// TIA Portal project "六路温湿度采集" (V16)

(* hardware
DEVICE "S71500/ET200MP station_1"  S7-1500 station
   slot 0: "导轨_0"  Rack  6ES7 590-1***0-0AA0
   slot 1: "PLC_1"  CPU 1512C-1 PN  6ES7 512-1CK01-0AB0  V2.8
      slot 3: "CPU 显示_1"  6ES7591-1AA00-0AA0
      slot 32768: "PROFINET 接口_1"  X1
         slot 32769: "端口_1"  X1 P1
         slot 32770: "端口_2"  X1 P2
      slot 34817: "Virtual CP interface port_1"  Virtual CP interface port  Virtual CP interface port
*)

// ===== PLC "PLC_1"  CPU 1512C-1 PN =====

VAR_GLOBAL   // PLC tag table "默认变量表"
   "中间变量" AT %MW100 : Word;
   "Tag_1" AT %M0.0 : Bool;
   "System_Byte" AT %MB1 : Byte;
   "FirstScan" AT %M1.0 : Bool;
   "DiagStatusUpdate" AT %M1.1 : Bool;
   "AlwaysTRUE" AT %M1.2 : Bool;
   "AlwaysFALSE" AT %M1.3 : Bool;
   "Tag_2" AT %M2.0 : Bool;
END_VAR

DATA_BLOCK "ModbusTCPData"   // DB1
{ S7_Optimized_Access := 'FALSE' }
VERSION : 0.1
   VAR
      模块1温度 : Int;
      模块1湿度 : Int;
      模块2温度 : Int;
      模块2湿度 : Int;
      模块3温度 : Int;
      模块3湿度 : Int;
      模块4温度 : Int;
      模块4湿度 : Int;
      模块5温度 : Int;
      模块5湿度 : Int;
      模块6温度 : Int;
      模块6湿度 : Int;
      模块1温度高 : Bool;
      模块1温度低 : Bool;
      模块1湿度高 : Bool;
      模块1湿度低 : Bool;
      模块1异常 : Bool;
      空1 : Bool;
      空2 : Bool;
      空3 : Bool;
      空byte1 : Byte;
      模块2温度高 : Bool;
      模块2温度低 : Bool;
      模块2湿度高 : Bool;
      模块2湿度低 : Bool;
      模块2异常 : Bool;
      空4 : Bool;
      空5 : Bool;
      空6 : Bool;
      空byte2 : Byte;
      模块3温度高 : Bool;
      模块3温度低 : Bool;
      模块3湿度高 : Bool;
      模块3湿度低 : Bool;
      模块3异常 : Bool;
      空7 : Bool;
      空8 : Bool;
      空9 : Bool;
      空byte3 : Byte;
      模块4温度高 : Bool;
      模块4温度低 : Bool;
      模块4湿度高 : Bool;
      模块4湿度低 : Bool;
      模块4异常 : Bool;
      空11 : Bool;
      空12 : Bool;
      空13 : Bool;
      空byte4 : Byte;
      模块5温度高 : Bool;
      模块5温度低 : Bool;
      模块5湿度高 : Bool;
      模块5湿度低 : Bool;
      模块5异常 : Bool;
      空14 : Bool;
      空15 : Bool;
      空16 : Bool;
      空byte5 : Byte;
      模块6温度高 : Bool;
      模块6温度低 : Bool;
      模块6湿度高 : Bool;
      模块6湿度低 : Bool;
      模块6异常 : Bool;
      空byte6 : Byte;
      模块1温度高限 : Int := 35;
      模块1温度低限 : Int := 25;
      模块1湿度高限 : Int := 25;
      模块1湿度低限 : Int := 15;
      模块2温度高限 : Int := 35;
      模块2温度低限 : Int := 25;
      模块2湿度高限 : Int := 25;
      模块2湿度低限 : Int := 15;
      模块3温度高限 : Int := 35;
      模块3温度低限 : Int := 25;
      模块3湿度高限 : Int := 25;
      模块3湿度低限 : Int := 15;
      模块4温度高限 : Int := 35;
      模块4温度低限 : Int := 25;
      模块4湿度高限 : Int := 25;
      模块4湿度低限 : Int := 15;
      模块5温度高限 : Int := 35;
      模块5温度低限 : Int := 25;
      模块5湿度高限 : Int := 25;
      模块5湿度低限 : Int := 15;
      模块6温度高限 : Int := 35;
      模块6温度低限 : Int := 25;
      模块6湿度高限 : Int := 25;
      模块6湿度低限 : Int := 15;
      模块1温度报警启用 : Int := 0;
      模块1湿度报警启用 : Int;
      模块2温度报警启用 : Int;
      模块2湿度报警启用 : Int;
      模块3温度报警启用 : Int;
      模块3湿度报警启用 : Int;
      模块4温度报警启用 : Int;
      模块4湿度报警启用 : Int;
      模块5温度报警启用 : Int;
      模块5湿度报警启用 : Int;
      模块6温度报警启用 : Int;
      模块6湿度报警启用 : Int;
      串口站地址 : Int;
      串口波特率 : Int;
      "IP地址-1" : Int;
      "IP地址-2" : Int;
      "IP地址-3" : Int;
      "IP地址-4" : Int;
      以太网端口号 : Int;
      "以太网参数写入确认（PC写1）" : Int;
   END_VAR
BEGIN
END_DATA_BLOCK

DATA_BLOCK "通信参数的DB块"   // DB3
{ S7_Optimized_Access := 'TRUE' }
VERSION : 0.1
   VAR
      Conn : TCON_IP_v4;
   END_VAR
BEGIN
   Conn.InterfaceId := 64;
   Conn.ID := 1;
   Conn.LocalPort := 502;
END_DATA_BLOCK

DATA_BLOCK "DateTime"   // DB4
{ S7_Optimized_Access := 'TRUE' }
VERSION : 0.1
   VAR
      day_time : DTL;
      ReadDateTIme_Now : Int;
   END_VAR
BEGIN
END_DATA_BLOCK

FUNCTION "温湿度模块超限报警" : Void   // FC1, LAD
{ S7_Optimized_Access := 'TRUE' }
VERSION : 0.1
   VAR_INPUT
      模块温度 : Int;
      模块温度高限 : Int;
      模块温度低限 : Int;
      模块湿度 : Int;
      模块湿度高限 : Int;
      模块湿度低限 : Int;
      模块温度报警启用 : Int;
      模块湿度报警启用 : Int;
   END_VAR
   VAR_OUTPUT
      模块异常 : Bool;
   END_VAR
   VAR_IN_OUT
      模块温度高 : Bool;
      模块温度低 : Bool;
      模块湿度高 : Bool;
      模块湿度低 : Bool;
   END_VAR
   VAR_TEMP   // added for the SCL form of the ladder/FBD networks
      _w1 : Bool;
      _w2 : Bool;
   END_VAR
BEGIN

REGION Network 1
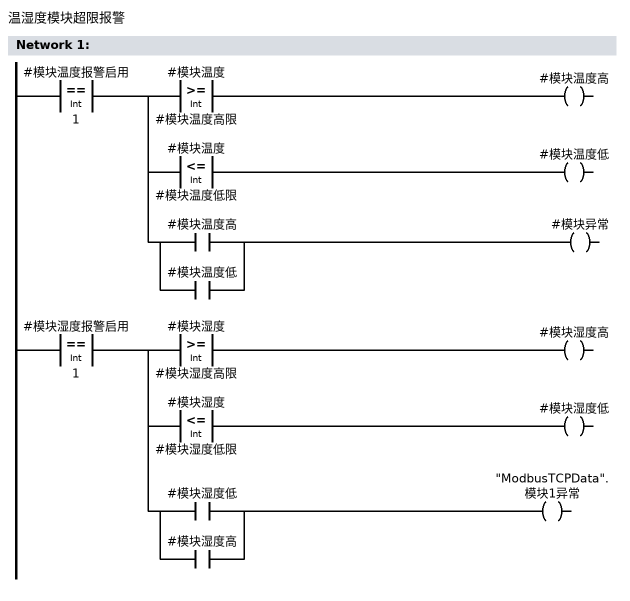
   RUNG wire#powerrail
      { S7_Templates := "SrcType := Int" } EQ_Contact(in1 := #模块温度报警启用, in2 := 1)
      wire#w1
      { S7_Templates := "SrcType := Int" } GE_Contact(in1 := #模块温度, in2 := #模块温度高限)
      Coil( #模块温度高 )
   END_RUNG
   RUNG wire#w1
      { S7_Templates := "SrcType := Int" } LE_Contact(in1 := #模块温度, in2 := #模块温度低限)
      Coil( #模块温度低 )
   END_RUNG
   RUNG wire#w1
      Contact( #模块温度高 )
      wire#w2
      Coil( #模块异常 )
   END_RUNG
   RUNG wire#w1
      Contact( #模块温度低 )
   END_RUNG wire#w2
   RUNG wire#powerrail
      { S7_Templates := "SrcType := Int" } EQ_Contact(in1 := #模块湿度报警启用, in2 := 1)
      wire#w3
      { S7_Templates := "SrcType := Int" } GE_Contact(in1 := #模块湿度, in2 := #模块湿度高限)
      Coil( #模块湿度高 )
   END_RUNG
   RUNG wire#w3
      { S7_Templates := "SrcType := Int" } LE_Contact(in1 := #模块湿度, in2 := #模块湿度低限)
      Coil( #模块湿度低 )
   END_RUNG
   RUNG wire#w3
      Contact( #模块湿度低 )
      wire#w4
      Coil( "ModbusTCPData".模块1异常 )
   END_RUNG
   RUNG wire#w3
      Contact( #模块湿度高 )
   END_RUNG wire#w4
   // the same network as SCL:
   #_w1 := #模块温度报警启用 = 1;
   #模块温度高 := #_w1 AND (#模块温度 >= #模块温度高限);
   #模块温度低 := #_w1 AND (#模块温度 <= #模块温度低限);
   #模块异常 := #_w1 AND (#模块温度高 OR #模块温度低);
   #_w2 := #模块湿度报警启用 = 1;
   #模块湿度高 := #_w2 AND (#模块湿度 >= #模块湿度高限);
   #模块湿度低 := #_w2 AND (#模块湿度 <= #模块湿度低限);
   "ModbusTCPData".模块1异常 := #_w2 AND (#模块湿度低 OR #模块湿度高);
END_REGION
END_FUNCTION

ORGANIZATION_BLOCK "Main"   // OB1, LAD, ProgramCycle
TITLE = "Main Program Sweep (Cycle)"
{ S7_Optimized_Access := 'TRUE' }
VERSION : 0.1
   VAR_INPUT
      Initial_Call : Bool;   // Initial call of this OB
      Remanence : Bool;   // =True, if remanent data are available
   END_VAR
BEGIN

REGION Network 1: 设定PLC的客户端，通信的变量
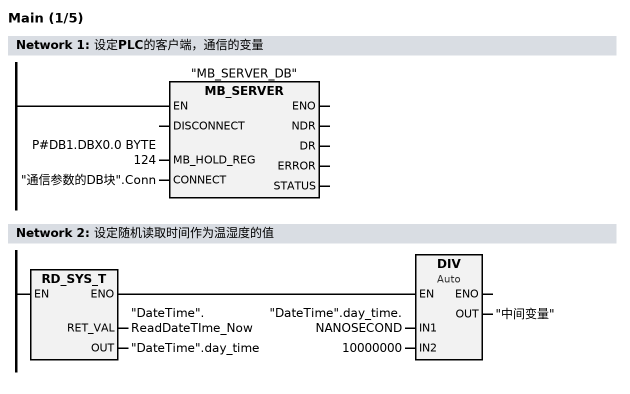
   "MB_SERVER_DB"(MB_HOLD_REG := P#DB1.DBX0.0 BYTE 124, CONNECT := "通信参数的DB块".Conn);   // MB_SERVER
END_REGION

REGION Network 2: 设定随机读取时间作为温湿度的值
   // ENO of a box is taken as its EN; it also drops when the box reports an error
   "DateTime".ReadDateTIme_Now := RD_SYS_T(OUT => "DateTime".day_time);
   "中间变量" := "DateTime".day_time.NANOSECOND / 10000000;
END_REGION

REGION Network 3: 将随机时间传递六路温湿度
   // 因为是毫秒机的显示，所以可以保证每个都不相同
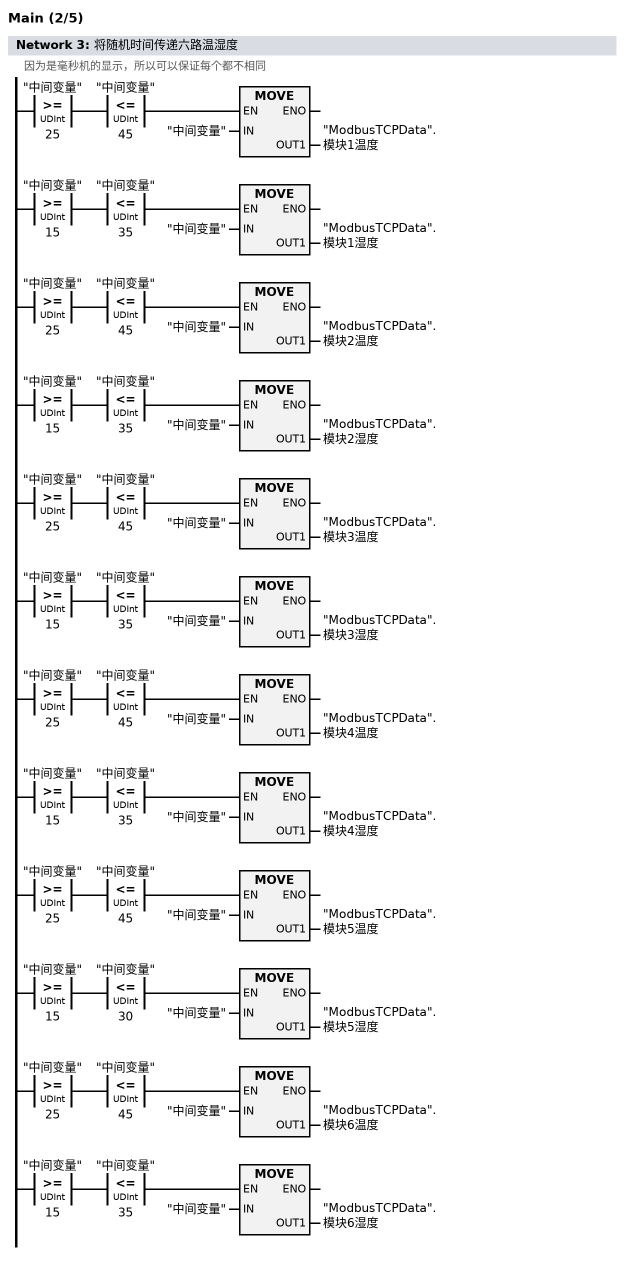
   RUNG wire#powerrail
      { S7_Templates := "SrcType := UDInt" } GE_Contact(in1 := "中间变量", in2 := 25)
      { S7_Templates := "SrcType := UDInt" } LE_Contact(in1 := "中间变量", in2 := 45)
      Move(in := "中间变量", out1 => "ModbusTCPData".模块1温度)
   END_RUNG
   RUNG wire#powerrail
      { S7_Templates := "SrcType := UDInt" } GE_Contact(in1 := "中间变量", in2 := 15)
      { S7_Templates := "SrcType := UDInt" } LE_Contact(in1 := "中间变量", in2 := 35)
      Move(in := "中间变量", out1 => "ModbusTCPData".模块1湿度)
   END_RUNG
   RUNG wire#powerrail
      { S7_Templates := "SrcType := UDInt" } GE_Contact(in1 := "中间变量", in2 := 25)
      { S7_Templates := "SrcType := UDInt" } LE_Contact(in1 := "中间变量", in2 := 45)
      Move(in := "中间变量", out1 => "ModbusTCPData".模块2温度)
   END_RUNG
   RUNG wire#powerrail
      { S7_Templates := "SrcType := UDInt" } GE_Contact(in1 := "中间变量", in2 := 15)
      { S7_Templates := "SrcType := UDInt" } LE_Contact(in1 := "中间变量", in2 := 35)
      Move(in := "中间变量", out1 => "ModbusTCPData".模块2湿度)
   END_RUNG
   RUNG wire#powerrail
      { S7_Templates := "SrcType := UDInt" } GE_Contact(in1 := "中间变量", in2 := 25)
      { S7_Templates := "SrcType := UDInt" } LE_Contact(in1 := "中间变量", in2 := 45)
      Move(in := "中间变量", out1 => "ModbusTCPData".模块3温度)
   END_RUNG
   RUNG wire#powerrail
      { S7_Templates := "SrcType := UDInt" } GE_Contact(in1 := "中间变量", in2 := 15)
      { S7_Templates := "SrcType := UDInt" } LE_Contact(in1 := "中间变量", in2 := 35)
      Move(in := "中间变量", out1 => "ModbusTCPData".模块3湿度)
   END_RUNG
   RUNG wire#powerrail
      { S7_Templates := "SrcType := UDInt" } GE_Contact(in1 := "中间变量", in2 := 25)
      { S7_Templates := "SrcType := UDInt" } LE_Contact(in1 := "中间变量", in2 := 45)
      Move(in := "中间变量", out1 => "ModbusTCPData".模块4温度)
   END_RUNG
   RUNG wire#powerrail
      { S7_Templates := "SrcType := UDInt" } GE_Contact(in1 := "中间变量", in2 := 15)
      { S7_Templates := "SrcType := UDInt" } LE_Contact(in1 := "中间变量", in2 := 35)
      Move(in := "中间变量", out1 => "ModbusTCPData".模块4湿度)
   END_RUNG
   RUNG wire#powerrail
      { S7_Templates := "SrcType := UDInt" } GE_Contact(in1 := "中间变量", in2 := 25)
      { S7_Templates := "SrcType := UDInt" } LE_Contact(in1 := "中间变量", in2 := 45)
      Move(in := "中间变量", out1 => "ModbusTCPData".模块5温度)
   END_RUNG
   RUNG wire#powerrail
      { S7_Templates := "SrcType := UDInt" } GE_Contact(in1 := "中间变量", in2 := 15)
      { S7_Templates := "SrcType := UDInt" } LE_Contact(in1 := "中间变量", in2 := 30)
      Move(in := "中间变量", out1 => "ModbusTCPData".模块5湿度)
   END_RUNG
   RUNG wire#powerrail
      { S7_Templates := "SrcType := UDInt" } GE_Contact(in1 := "中间变量", in2 := 25)
      { S7_Templates := "SrcType := UDInt" } LE_Contact(in1 := "中间变量", in2 := 45)
      Move(in := "中间变量", out1 => "ModbusTCPData".模块6温度)
   END_RUNG
   RUNG wire#powerrail
      { S7_Templates := "SrcType := UDInt" } GE_Contact(in1 := "中间变量", in2 := 15)
      { S7_Templates := "SrcType := UDInt" } LE_Contact(in1 := "中间变量", in2 := 35)
      Move(in := "中间变量", out1 => "ModbusTCPData".模块6湿度)
   END_RUNG
   // the same network as SCL:
   IF ("中间变量" >= 25) AND ("中间变量" <= 45) THEN "ModbusTCPData".模块1温度 := "中间变量"; END_IF;
   IF ("中间变量" >= 15) AND ("中间变量" <= 35) THEN "ModbusTCPData".模块1湿度 := "中间变量"; END_IF;
   IF ("中间变量" >= 25) AND ("中间变量" <= 45) THEN "ModbusTCPData".模块2温度 := "中间变量"; END_IF;
   IF ("中间变量" >= 15) AND ("中间变量" <= 35) THEN "ModbusTCPData".模块2湿度 := "中间变量"; END_IF;
   IF ("中间变量" >= 25) AND ("中间变量" <= 45) THEN "ModbusTCPData".模块3温度 := "中间变量"; END_IF;
   IF ("中间变量" >= 15) AND ("中间变量" <= 35) THEN "ModbusTCPData".模块3湿度 := "中间变量"; END_IF;
   IF ("中间变量" >= 25) AND ("中间变量" <= 45) THEN "ModbusTCPData".模块4温度 := "中间变量"; END_IF;
   IF ("中间变量" >= 15) AND ("中间变量" <= 35) THEN "ModbusTCPData".模块4湿度 := "中间变量"; END_IF;
   IF ("中间变量" >= 25) AND ("中间变量" <= 45) THEN "ModbusTCPData".模块5温度 := "中间变量"; END_IF;
   IF ("中间变量" >= 15) AND ("中间变量" <= 30) THEN "ModbusTCPData".模块5湿度 := "中间变量"; END_IF;
   IF ("中间变量" >= 25) AND ("中间变量" <= 45) THEN "ModbusTCPData".模块6温度 := "中间变量"; END_IF;
   IF ("中间变量" >= 15) AND ("中间变量" <= 35) THEN "ModbusTCPData".模块6湿度 := "中间变量"; END_IF;
END_REGION

REGION Network 4
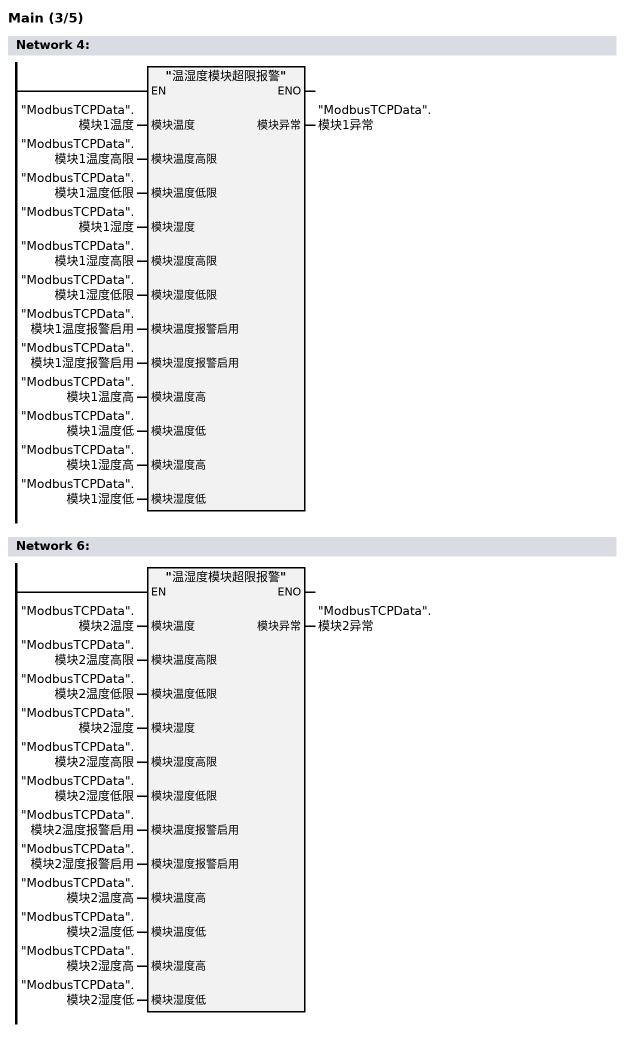
   RUNG wire#powerrail
      "温湿度模块超限报警"(模块温度 := "ModbusTCPData".模块1温度, 模块温度高限 := "ModbusTCPData".模块1温度高限, 模块温度低限 := "ModbusTCPData".模块1温度低限, 模块湿度 := "ModbusTCPData".模块1湿度, 模块湿度高限 := "ModbusTCPData".模块1湿度高限, 模块湿度低限 := "ModbusTCPData".模块1湿度低限, 模块温度报警启用 := "ModbusTCPData".模块1温度报警启用, 模块湿度报警启用 := "ModbusTCPData".模块1湿度报警启用, 模块温度高 := "ModbusTCPData".模块1温度高, 模块温度低 := "ModbusTCPData".模块1温度低, 模块湿度高 := "ModbusTCPData".模块1湿度高, 模块湿度低 := "ModbusTCPData".模块1湿度低, 模块异常 => "ModbusTCPData".模块1异常)
   END_RUNG
   // the same network as SCL:
   "温湿度模块超限报警"(模块温度 := "ModbusTCPData".模块1温度,
               模块温度高限 := "ModbusTCPData".模块1温度高限,
               模块温度低限 := "ModbusTCPData".模块1温度低限,
               模块湿度 := "ModbusTCPData".模块1湿度,
               模块湿度高限 := "ModbusTCPData".模块1湿度高限,
               模块湿度低限 := "ModbusTCPData".模块1湿度低限,
               模块温度报警启用 := "ModbusTCPData".模块1温度报警启用,
               模块湿度报警启用 := "ModbusTCPData".模块1湿度报警启用,
               模块温度高 := "ModbusTCPData".模块1温度高,
               模块温度低 := "ModbusTCPData".模块1温度低,
               模块湿度高 := "ModbusTCPData".模块1湿度高,
               模块湿度低 := "ModbusTCPData".模块1湿度低,
               模块异常 => "ModbusTCPData".模块1异常);
END_REGION

REGION Network 6
   RUNG wire#powerrail
      "温湿度模块超限报警"(模块温度 := "ModbusTCPData".模块2温度, 模块温度高限 := "ModbusTCPData".模块2温度高限, 模块温度低限 := "ModbusTCPData".模块2温度低限, 模块湿度 := "ModbusTCPData".模块2湿度, 模块湿度高限 := "ModbusTCPData".模块2湿度高限, 模块湿度低限 := "ModbusTCPData".模块2湿度低限, 模块温度报警启用 := "ModbusTCPData".模块2温度报警启用, 模块湿度报警启用 := "ModbusTCPData".模块2湿度报警启用, 模块温度高 := "ModbusTCPData".模块2温度高, 模块温度低 := "ModbusTCPData".模块2温度低, 模块湿度高 := "ModbusTCPData".模块2湿度高, 模块湿度低 := "ModbusTCPData".模块2湿度低, 模块异常 => "ModbusTCPData".模块2异常)
   END_RUNG
   // the same network as SCL:
   "温湿度模块超限报警"(模块温度 := "ModbusTCPData".模块2温度,
               模块温度高限 := "ModbusTCPData".模块2温度高限,
               模块温度低限 := "ModbusTCPData".模块2温度低限,
               模块湿度 := "ModbusTCPData".模块2湿度,
               模块湿度高限 := "ModbusTCPData".模块2湿度高限,
               模块湿度低限 := "ModbusTCPData".模块2湿度低限,
               模块温度报警启用 := "ModbusTCPData".模块2温度报警启用,
               模块湿度报警启用 := "ModbusTCPData".模块2湿度报警启用,
               模块温度高 := "ModbusTCPData".模块2温度高,
               模块温度低 := "ModbusTCPData".模块2温度低,
               模块湿度高 := "ModbusTCPData".模块2湿度高,
               模块湿度低 := "ModbusTCPData".模块2湿度低,
               模块异常 => "ModbusTCPData".模块2异常);
END_REGION

REGION Network 7
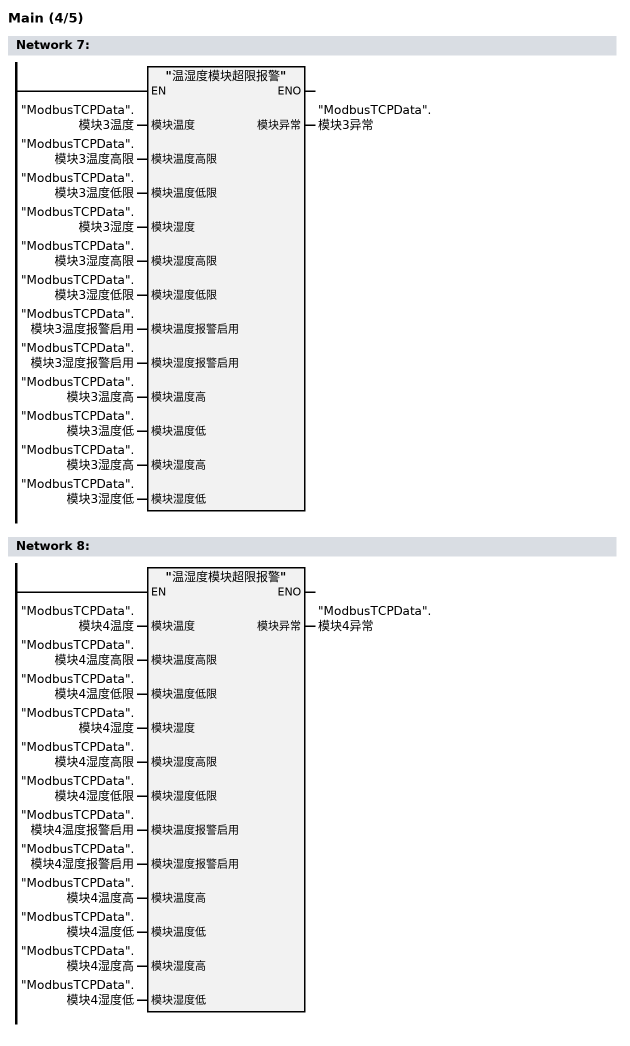
   RUNG wire#powerrail
      "温湿度模块超限报警"(模块温度 := "ModbusTCPData".模块3温度, 模块温度高限 := "ModbusTCPData".模块3温度高限, 模块温度低限 := "ModbusTCPData".模块3温度低限, 模块湿度 := "ModbusTCPData".模块3湿度, 模块湿度高限 := "ModbusTCPData".模块3湿度高限, 模块湿度低限 := "ModbusTCPData".模块3湿度低限, 模块温度报警启用 := "ModbusTCPData".模块3温度报警启用, 模块湿度报警启用 := "ModbusTCPData".模块3湿度报警启用, 模块温度高 := "ModbusTCPData".模块3温度高, 模块温度低 := "ModbusTCPData".模块3温度低, 模块湿度高 := "ModbusTCPData".模块3湿度高, 模块湿度低 := "ModbusTCPData".模块3湿度低, 模块异常 => "ModbusTCPData".模块3异常)
   END_RUNG
   // the same network as SCL:
   "温湿度模块超限报警"(模块温度 := "ModbusTCPData".模块3温度,
               模块温度高限 := "ModbusTCPData".模块3温度高限,
               模块温度低限 := "ModbusTCPData".模块3温度低限,
               模块湿度 := "ModbusTCPData".模块3湿度,
               模块湿度高限 := "ModbusTCPData".模块3湿度高限,
               模块湿度低限 := "ModbusTCPData".模块3湿度低限,
               模块温度报警启用 := "ModbusTCPData".模块3温度报警启用,
               模块湿度报警启用 := "ModbusTCPData".模块3湿度报警启用,
               模块温度高 := "ModbusTCPData".模块3温度高,
               模块温度低 := "ModbusTCPData".模块3温度低,
               模块湿度高 := "ModbusTCPData".模块3湿度高,
               模块湿度低 := "ModbusTCPData".模块3湿度低,
               模块异常 => "ModbusTCPData".模块3异常);
END_REGION

REGION Network 8
   RUNG wire#powerrail
      "温湿度模块超限报警"(模块温度 := "ModbusTCPData".模块4温度, 模块温度高限 := "ModbusTCPData".模块4温度高限, 模块温度低限 := "ModbusTCPData".模块4温度低限, 模块湿度 := "ModbusTCPData".模块4湿度, 模块湿度高限 := "ModbusTCPData".模块4湿度高限, 模块湿度低限 := "ModbusTCPData".模块4湿度低限, 模块温度报警启用 := "ModbusTCPData".模块4温度报警启用, 模块湿度报警启用 := "ModbusTCPData".模块4湿度报警启用, 模块温度高 := "ModbusTCPData".模块4温度高, 模块温度低 := "ModbusTCPData".模块4温度低, 模块湿度高 := "ModbusTCPData".模块4湿度高, 模块湿度低 := "ModbusTCPData".模块4湿度低, 模块异常 => "ModbusTCPData".模块4异常)
   END_RUNG
   // the same network as SCL:
   "温湿度模块超限报警"(模块温度 := "ModbusTCPData".模块4温度,
               模块温度高限 := "ModbusTCPData".模块4温度高限,
               模块温度低限 := "ModbusTCPData".模块4温度低限,
               模块湿度 := "ModbusTCPData".模块4湿度,
               模块湿度高限 := "ModbusTCPData".模块4湿度高限,
               模块湿度低限 := "ModbusTCPData".模块4湿度低限,
               模块温度报警启用 := "ModbusTCPData".模块4温度报警启用,
               模块湿度报警启用 := "ModbusTCPData".模块4湿度报警启用,
               模块温度高 := "ModbusTCPData".模块4温度高,
               模块温度低 := "ModbusTCPData".模块4温度低,
               模块湿度高 := "ModbusTCPData".模块4湿度高,
               模块湿度低 := "ModbusTCPData".模块4湿度低,
               模块异常 => "ModbusTCPData".模块4异常);
END_REGION

REGION Network 9
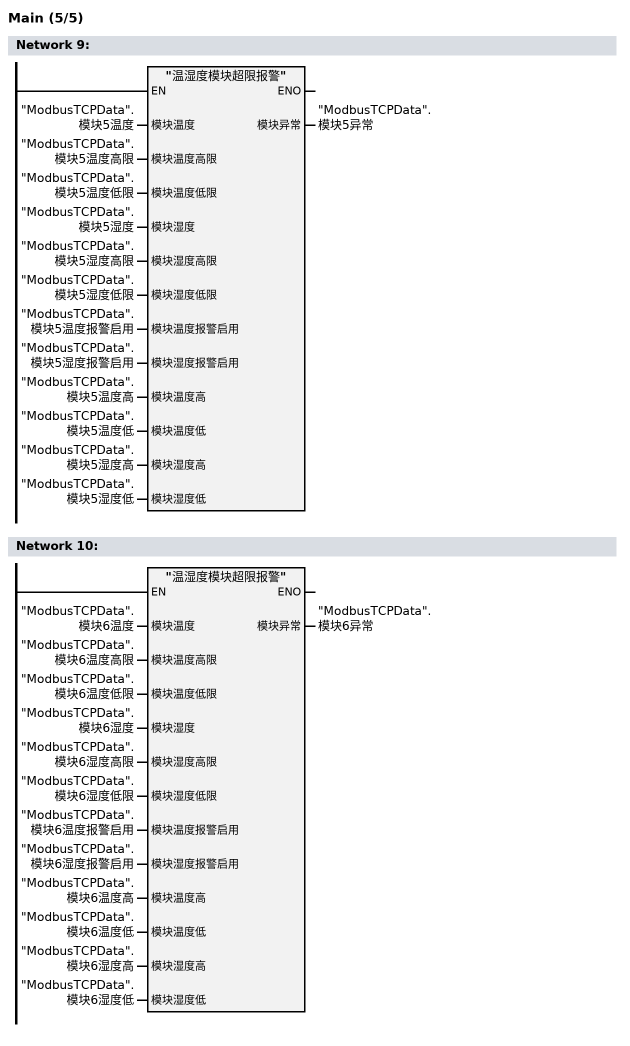
   RUNG wire#powerrail
      "温湿度模块超限报警"(模块温度 := "ModbusTCPData".模块5温度, 模块温度高限 := "ModbusTCPData".模块5温度高限, 模块温度低限 := "ModbusTCPData".模块5温度低限, 模块湿度 := "ModbusTCPData".模块5湿度, 模块湿度高限 := "ModbusTCPData".模块5湿度高限, 模块湿度低限 := "ModbusTCPData".模块5湿度低限, 模块温度报警启用 := "ModbusTCPData".模块5温度报警启用, 模块湿度报警启用 := "ModbusTCPData".模块5湿度报警启用, 模块温度高 := "ModbusTCPData".模块5温度高, 模块温度低 := "ModbusTCPData".模块5温度低, 模块湿度高 := "ModbusTCPData".模块5湿度高, 模块湿度低 := "ModbusTCPData".模块5湿度低, 模块异常 => "ModbusTCPData".模块5异常)
   END_RUNG
   // the same network as SCL:
   "温湿度模块超限报警"(模块温度 := "ModbusTCPData".模块5温度,
               模块温度高限 := "ModbusTCPData".模块5温度高限,
               模块温度低限 := "ModbusTCPData".模块5温度低限,
               模块湿度 := "ModbusTCPData".模块5湿度,
               模块湿度高限 := "ModbusTCPData".模块5湿度高限,
               模块湿度低限 := "ModbusTCPData".模块5湿度低限,
               模块温度报警启用 := "ModbusTCPData".模块5温度报警启用,
               模块湿度报警启用 := "ModbusTCPData".模块5湿度报警启用,
               模块温度高 := "ModbusTCPData".模块5温度高,
               模块温度低 := "ModbusTCPData".模块5温度低,
               模块湿度高 := "ModbusTCPData".模块5湿度高,
               模块湿度低 := "ModbusTCPData".模块5湿度低,
               模块异常 => "ModbusTCPData".模块5异常);
END_REGION

REGION Network 10
   RUNG wire#powerrail
      "温湿度模块超限报警"(模块温度 := "ModbusTCPData".模块6温度, 模块温度高限 := "ModbusTCPData".模块6温度高限, 模块温度低限 := "ModbusTCPData".模块6温度低限, 模块湿度 := "ModbusTCPData".模块6湿度, 模块湿度高限 := "ModbusTCPData".模块6湿度高限, 模块湿度低限 := "ModbusTCPData".模块6湿度低限, 模块温度报警启用 := "ModbusTCPData".模块6温度报警启用, 模块湿度报警启用 := "ModbusTCPData".模块6湿度报警启用, 模块温度高 := "ModbusTCPData".模块6温度高, 模块温度低 := "ModbusTCPData".模块6温度低, 模块湿度高 := "ModbusTCPData".模块6湿度高, 模块湿度低 := "ModbusTCPData".模块6湿度低, 模块异常 => "ModbusTCPData".模块6异常)
   END_RUNG
   // the same network as SCL:
   "温湿度模块超限报警"(模块温度 := "ModbusTCPData".模块6温度,
               模块温度高限 := "ModbusTCPData".模块6温度高限,
               模块温度低限 := "ModbusTCPData".模块6温度低限,
               模块湿度 := "ModbusTCPData".模块6湿度,
               模块湿度高限 := "ModbusTCPData".模块6湿度高限,
               模块湿度低限 := "ModbusTCPData".模块6湿度低限,
               模块温度报警启用 := "ModbusTCPData".模块6温度报警启用,
               模块湿度报警启用 := "ModbusTCPData".模块6湿度报警启用,
               模块温度高 := "ModbusTCPData".模块6温度高,
               模块温度低 := "ModbusTCPData".模块6温度低,
               模块湿度高 := "ModbusTCPData".模块6湿度高,
               模块湿度低 := "ModbusTCPData".模块6湿度低,
               模块异常 => "ModbusTCPData".模块6异常);
END_REGION
END_ORGANIZATION_BLOCK